// Mitsubishi GX Works2 project: Auto reverse forward   PLC: FX1N/FX1NC

PROGRAM MAIN
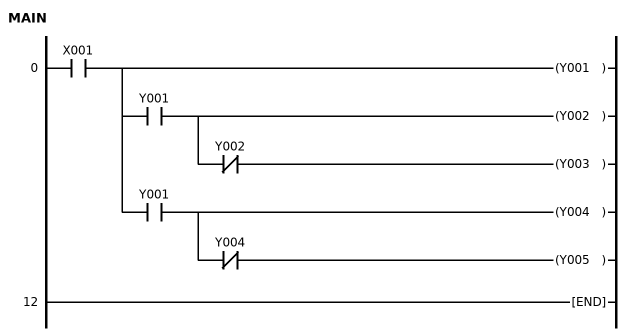
0     LD      X001
      OUT     Y001
      MPS
      AND     Y001
      OUT     Y002
      ANI     Y002
      OUT     Y003
      MPP
      AND     Y001
      OUT     Y004
      ANI     Y004
      OUT     Y005
12    END
END_PROGRAM
